// TwinCAT 3 PLC project PLC1
// ProgramVersion: 3.1.4024.12
// libraries:
//   Tc2_Standard, * (Beckhoff Automation GmbH)
//   Tc2_System, * (Beckhoff Automation GmbH)
//   Tc3_Module, * (Beckhoff Automation GmbH)
// project tree:
//   Diagrams/ Class Diagram.TcCD (not stored)
//   FBs/ FB_Generator.TcPOU, FB_GeneratorEX.TcPOU
//   / PlcTask.TcTTO
//   POUs/ MAIN.TcPOU
// real-time tasks:
//   TASK PlcTask: cycle T#10ms, priority 20, ADS port 350

CONFIGURATION PLC1
    RESOURCE PLC ON TwinCAT3
        TASK PlcTask(INTERVAL := T#10ms, PRIORITY := 20);
        PROGRAM MAIN WITH PlcTask : MAIN;
    END_RESOURCE
END_CONFIGURATION

// ---- POUs/MAIN.TcPOU
PROGRAM MAIN
VAR
	// Instance of Generator 1
	fbGenerator1 :FB_Generator;	
	// Instance of Generator 2
	fbGenerator2 :FB_GeneratorEX;	
	
	// Status of flasher 1
	Flasher1: BOOL;
	// Status of flasher 2
	Flasher2: BOOL;
END_VAR

// Set the cycletime property for the class
fbGenerator1.Cycletime := T#2S;
fbGenerator2.Cycletime := T#2S;

// Call the flasher method
Flasher1 := fbGenerator1.Flash();
Flasher2 := fbGenerator2.Flash();

END_PROGRAM

// ---- FBs/FB_Generator.TcPOU
FUNCTION_BLOCK FB_Generator
VAR_INPUT
END_VAR
VAR_OUTPUT
END_VAR
VAR
	// instance variables
	fbTon1		: TON;	
	tCycletime	: TIME:=T#1S;
	bToggle		: BOOL;

	
	fbTp1		: TP;		
	tPulsetime	: TIME := T#800MS;
END_VAR

PROPERTY Cycletime : TIME
GET
Cycletime := this^.tCycletime;
END_GET
SET
(*Limit Input Value *)
IF Cycletime < T#50MS THEN
	tCycletime := T#50MS;
ELSIF Cycletime > T#5S THEN
	tCycletime := T#5S;
ELSE	
	tCycletime := Cycletime;
END_IF
END_SET
END_PROPERTY

METHOD Flash : BOOL
VAR_INPUT
END_VAR
fbTon1(IN:= NOT fbTon1.Q , PT:=THIS^.tCycletime , Q=> , ET=> );
IF fbTon1.Q THEN
	bToggle:= NOT bToggle;
END_IF
Flash:= bToggle;
END_METHOD

METHOD Pulse : BOOL
VAR_INPUT
	bTriggPuls: BOOL;
END_VAR
fbTp1(IN:=bTriggPuls , PT:=this^.tPulsetime , Q=>Pulse , ET=> );
END_METHOD

PROPERTY Vendor : STRING
GET
Vendor := 'Training';
END_GET
END_PROPERTY

END_FUNCTION_BLOCK

// ---- FBs/FB_GeneratorEX.TcPOU
FUNCTION_BLOCK FB_GeneratorEX EXTENDS FB_Generator
VAR_INPUT
END_VAR
VAR_OUTPUT
END_VAR
VAR
END_VAR

METHOD Flash : BOOL
VAR_INPUT
END_VAR
fbTon1(IN:=NOT fbTon1.Q , PT:= 2* tCycletime , Q=> , ET=> );
Flash := fbTon1.ET < fbTon1.PT / 3;
END_METHOD

PROPERTY Vendor : STRING
GET
Vendor := CONCAT
			(
			STR1:= 'Company b, based on' , 
			STR2:=SUPER^.Vendor 
			);
END_GET
END_PROPERTY

END_FUNCTION_BLOCK
